PROGRAM nN_coeff_calculation
VAR
	I: WORD;//loop  variable
	
	power_accumulated_run: REAL := 0;// Auxiliar accumulator
	
END_VAR

(*
***************************************************************************************************
* \file    nN coefficient calculation
* \author  Quique
* \version V1.0.0
* \date    12/08/2022
* \brief   Calculation of n/N coefficient
***************************************************************************************************

\brief   Code block used to calculate n/N coefficient for converters running

\details	This code looks which inverters are online and running (on state), understanding
			that those inverters are controllable by PPC. Then it takes the power of those
			controlable ones, sums it and compares with plant nominal power to obtain a 
			coefficient of the inverters' powers running and able to control with respect to 
			plant total.  
	     
*)

FOR I := 1 TO GVL_CONV_COMMS.NUMBER_CONVERTERS DO;
	
	IF GVL_CONV_COMMS.Current_Status[I] = GVL_CONVERTERS_COMMON.CONVERTER_STATUS_RUN AND GVL_CONV_COMMS.ERROR_TASK[I] <> 1 THEN
		//Only inverters in ON status and online are taken into account
		power_accumulated_run := power_accumulated_run + GVL_CONV_COMMS.CONVERTERS[I].Capacity;
	END_IF
END_FOR

GVL_CONV_COMMS.converters_nN_coeff := power_accumulated_run / GVL_PLANT_DEF.Plant_capacity_nom;
power_accumulated_run := 0;

END_PROGRAM

(* stored: Version 1.1.0.1, ProductVersion 3.1.4024.11
   POU nN_coeff_calculation: Id {76a51f9a-789b-4048-a626-a8e3ed805077}, SpecialFunc None *)
